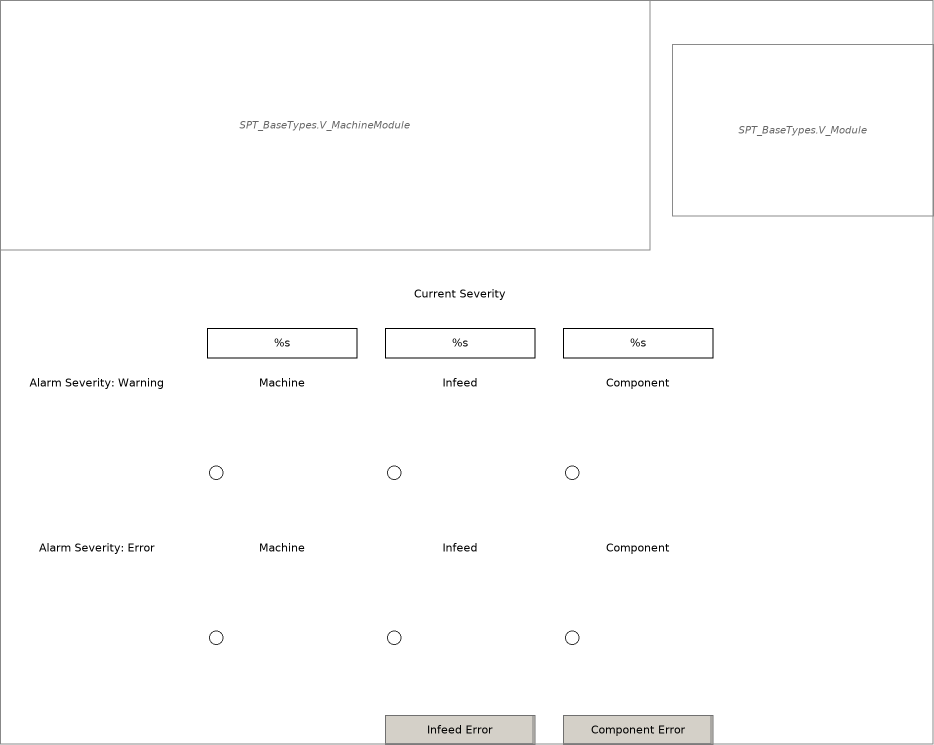
VISUALIZATION Visualization  // 934x745
    Frame (0,0 650x250)
        shows SPT_BaseTypes.V_MachineModule(HMI := MAIN.Machine.PackMLBaseModule_HMI)
    Label (207,533 150x30), "Machine"
    Label (385,533 150x30), "Infeed"
    Label (563,533 150x30), "Component"
    Label (22,533 150x30), "Alarm Severity: Error"
    RadioButton (207,584 168x107), variable: MAIN.Machine._ErrorSeverity
        Areas[0]: Text=Warning
        Areas[1]: Text=Abort Immediate
        Areas[2]: Text=Abort Immediate Error
    RadioButton (385,584 168x107), variable: MAIN.Machine.Infeed._ErrorSeverity
        Areas[0]: Text=Warning
        Areas[1]: Text=Abort Immediate
        Areas[2]: Text=Abort Immediate Error
    RadioButton (563,584 168x107), variable: MAIN.Machine.Infeed.Component._ErrorSeverity
        Areas[0]: Text=Warning
        Areas[1]: Text=Abort Immediate
        Areas[2]: Text=Abort Immediate Error
    Button (563,715 150x30), "Component Error"
        toggle MAIN.Machine.Infeed.Component.testError
    Frame (672,44 262x172)
        shows SPT_BaseTypes.V_Module(HMI := MAIN.Machine.Infeed.PackMLBaseModule_HMI)
    Button (385,715 150x30), "Infeed Error"
        toggle MAIN.Machine.Infeed.testError
    Label (207,368 150x30), "Machine"
    Label (385,368 150x30), "Infeed"
    Label (563,368 150x30), "Component"
    Label (22,368 150x30), "Alarm Severity: Warning"
    RadioButton (207,419 168x107), variable: MAIN.Machine._WarningSeverity
        Areas[0]: Text=Warning
        Areas[1]: Text=Abort Immediate
        Areas[2]: Text=Abort Immediate Error
    RadioButton (385,419 168x107), variable: MAIN.Machine.Infeed._WarningSeverity
        Areas[0]: Text=Warning
        Areas[1]: Text=Abort Immediate
        Areas[2]: Text=Abort Immediate Error
    RadioButton (563,419 168x107), variable: MAIN.Machine.Infeed.Component._WarningSeverity
        Areas[0]: Text=Warning
        Areas[1]: Text=Abort Immediate
        Areas[2]: Text=Abort Immediate Error
    Rectangle (207,328 150x30), "%s", text variable: MAIN.Machine._CurrentAlarmSeverity
    Rectangle (385,328 150x30), "%s", text variable: MAIN.Machine.Infeed._CurrentAlarmSeverity
    Rectangle (563,328 150x30), "%s", text variable: MAIN.Machine.Infeed.Component._CurrentAlarmSeverity
    Label (385,279 150x30), "Current Severity"
END_VISUALIZATION

(* stored: Version 1.1.0.1
   Visu Visualization: Id {9c99bfbb-2717-4adc-9050-115bd62bf7c8} *)
